# EPICS substitutions: template/evr-cpci-230-ess.substitutions
# Record set for a cPCI-EVR-230
#
# Macros:
#  OBJ = Card name (same as mrmEvrSetupPCI())
#  P and R = System and Device name
#  FEVT = Event link frequency (default 88.0525 MHz)
#
# Record names have the general forms:
#  $(P)$(R=)$(S=:)Signal-SD
#  $(P)$(R=)$(S=:)SubDev-Signal-SD

file "mrmevrbase.template"
{
{P="\$(P)\$(R=)\$(S=:)", PSRC="\$(P)\$(R=)\$(S=:)Src-", PCNT="\$(P)\$(R=)\$(S=:)Cnt-", PLINK="\$(P)\$(R=)\$(S=:)Link-", PRATE="\$(P)\$(R=)\$(S=:)Rate-", PTIME="\$(P)\$(R=)\$(S=:)Time-", OBJ="\$(OBJ)", OBJBUFRX="\$(OBJ):BUFRX", EVNT1HZ="\$(EVNT1HZ=125)", FEVT="\$(FEVT=88.0525)"}
}

file "databuftx.db"
{pattern
{P, OBJ, PROTO}
{"\$(P)\$(R=)\$(S=:)dbus-send-", "\$(OBJ):BUFTX", 1}
}

file "databuftxCtrl.db"
{pattern
{P, OBJ}
{"\$(P)\$(R=)\$(S=:)Link-", "\$(OBJ):BUFTX"}
}

file "mrmevrbufrx.db"
{pattern
{P, OBJ, PROTO}
{"\$(P)\$(R=)\$(S=:)dbus-recv-", \$(OBJ):BUFRX, 0xff00}
}

file "sfp.db"
{
{P="\$(P)\$(R=)\$(S=:)SFP-", PPWR="\$(P)\$(R=)\$(S=:)SFP-Pwr-", PSPEED="\$(P)\$(R=)\$(S=:)SFP-Speed-", PDATE="\$(P)\$(R=)\$(S=:)SFP-Date-", OBJ="\$(OBJ):SFP"}
}

file "evrmap.db"
{pattern
{NAME, OBJ, func, EVT}
{"\$(P)\$(R=)\$(S=:)Evt-Blink0-SP", "\$(OBJ)", Blink, 15}
{"\$(P)\$(R=)\$(S=:)Evt-Blink1-SP", "\$(OBJ)", Blink, 0}
{"\$(P)\$(R=)\$(S=:)Evt-ResetPS-SP","\$(OBJ)", "Reset PS", 123}
}

file "evrevent.db"
{pattern
{EN, OBJ, CODE, EVNT}
{"\$(P)\$(R=)\$(S=:)1hz",  "\$(OBJ)", 0x7d, 125}
{"\$(P)\$(R=)\$(S=:)EvtA", "\$(OBJ)", 10, 10}
{"\$(P)\$(R=)\$(S=:)EvtB", "\$(OBJ)", 11, 11}
{"\$(P)\$(R=)\$(S=:)EvtC", "\$(OBJ)", 12, 12}
{"\$(P)\$(R=)\$(S=:)EvtD", "\$(OBJ)", 13, 13}
{"\$(P)\$(R=)\$(S=:)EvtE", "\$(OBJ)", 14, 14}
{"\$(P)\$(R=)\$(S=:)EvtF", "\$(OBJ)", 15, 15}
{"\$(P)\$(R=)\$(S=:)EvtG", "\$(OBJ)", 16, 16}
{"\$(P)\$(R=)\$(S=:)EvtH", "\$(OBJ)", 17, 17}
}

file "evrscale.db"
{pattern
{IDX, P, SN, OBJ, MAX}
{0, "\$(P)\$(R=)\$(S=:)Link-", "\$(P)\$(R=)\$(S=:)PS$(IDX)-", "\$(OBJ):PS$(IDX)", "0xffffffff"}
{1, "\$(P)\$(R=)\$(S=:)Link-", "\$(P)\$(R=)\$(S=:)PS$(IDX)-", "\$(OBJ):PS$(IDX)", "0xffffffff"}
{2, "\$(P)\$(R=)\$(S=:)Link-", "\$(P)\$(R=)\$(S=:)PS$(IDX)-", "\$(OBJ):PS$(IDX)", "0xffffffff"}
}

file "mrmevrout.db"
{pattern
{ON, ONSRC, OBJ, DESC}
{"\$(P)\$(R=)\$(S=:)OutInt-", "\$(P)\$(R=)\$(S=:)OutInt-Src-", "\$(OBJ):Int", "Internal"}
{"\$(P)\$(R=)\$(S=:)OutFPUV0-", "\$(P)\$(R=)\$(S=:)OutFPUV0-Src-", "\$(OBJ):FrontUnivOut0", "UNIV0"}
{"\$(P)\$(R=)\$(S=:)OutFPUV1-", "\$(P)\$(R=)\$(S=:)OutFPUV1-Src-", "\$(OBJ):FrontUnivOut1", "UNIV1"}
{"\$(P)\$(R=)\$(S=:)OutFPUV2-", "\$(P)\$(R=)\$(S=:)OutFPUV2-Src-", "\$(OBJ):FrontUnivOut2", "UNIV2"}
{"\$(P)\$(R=)\$(S=:)OutFPUV3-", "\$(P)\$(R=)\$(S=:)OutFPUV3-Src-", "\$(OBJ):FrontUnivOut3", "UNIV3"}
}

file "mrmevroutint.db"
{{
    ON="\$(P)\$(R=)\$(S=:)OutInt-", OBJ="\$(OBJ)"
}}

# Pulse generators w/o a prescaler set NOPS=1
file "evrpulser.db"
{pattern
{PID, P, PLINK, PN, PNDELAY, PNWIDTH, OBJ, DMAX, WMAX, PMAX, NOPS}
{0, "\$(P)\$(R=)\$(S=:)", "\$(P)\$(R=)\$(S=:)Link-", "\$(P)\$(R=)\$(S=:)DlyGen$(PID)-", "\$(P)\$(R=)\$(S=:)DlyGen$(PID)-Delay-", "\$(P)\$(R=)\$(S=:)DlyGen$(PID)-Width-", "\$(OBJ):Pul$(PID)", "0xffffffff", "0xffffffff", "0xffff", 0}
{1, "\$(P)\$(R=)\$(S=:)", "\$(P)\$(R=)\$(S=:)Link-", "\$(P)\$(R=)\$(S=:)DlyGen$(PID)-", "\$(P)\$(R=)\$(S=:)DlyGen$(PID)-Delay-", "\$(P)\$(R=)\$(S=:)DlyGen$(PID)-Width-", "\$(OBJ):Pul$(PID)", "0xffffffff", "0xffffffff", "0xffff", 0}
{2, "\$(P)\$(R=)\$(S=:)", "\$(P)\$(R=)\$(S=:)Link-", "\$(P)\$(R=)\$(S=:)DlyGen$(PID)-", "\$(P)\$(R=)\$(S=:)DlyGen$(PID)-Delay-", "\$(P)\$(R=)\$(S=:)DlyGen$(PID)-Width-", "\$(OBJ):Pul$(PID)", "0xffffffff", "0xffffffff", "0xffff", 0}
{3, "\$(P)\$(R=)\$(S=:)", "\$(P)\$(R=)\$(S=:)Link-", "\$(P)\$(R=)\$(S=:)DlyGen$(PID)-", "\$(P)\$(R=)\$(S=:)DlyGen$(PID)-Delay-", "\$(P)\$(R=)\$(S=:)DlyGen$(PID)-Width-", "\$(OBJ):Pul$(PID)", "0xffffffff", "0xffffffff", "0xffff", 0}
{4, "\$(P)\$(R=)\$(S=:)", "\$(P)\$(R=)\$(S=:)Link-", "\$(P)\$(R=)\$(S=:)DlyGen$(PID)-", "\$(P)\$(R=)\$(S=:)DlyGen$(PID)-Delay-", "\$(P)\$(R=)\$(S=:)DlyGen$(PID)-Width-", "\$(OBJ):Pul$(PID)", "0xffffffff", "0xffff", "1", 1}
{5, "\$(P)\$(R=)\$(S=:)", "\$(P)\$(R=)\$(S=:)Link-", "\$(P)\$(R=)\$(S=:)DlyGen$(PID)-", "\$(P)\$(R=)\$(S=:)DlyGen$(PID)-Delay-", "\$(P)\$(R=)\$(S=:)DlyGen$(PID)-Width-", "\$(OBJ):Pul$(PID)", "0xffffffff", "0xffff", "1", 1}
{6, "\$(P)\$(R=)\$(S=:)", "\$(P)\$(R=)\$(S=:)Link-", "\$(P)\$(R=)\$(S=:)DlyGen$(PID)-", "\$(P)\$(R=)\$(S=:)DlyGen$(PID)-Delay-", "\$(P)\$(R=)\$(S=:)DlyGen$(PID)-Width-", "\$(OBJ):Pul$(PID)", "0xffffffff", "0xffff", "1", 1}
{7, "\$(P)\$(R=)\$(S=:)", "\$(P)\$(R=)\$(S=:)Link-", "\$(P)\$(R=)\$(S=:)DlyGen$(PID)-", "\$(P)\$(R=)\$(S=:)DlyGen$(PID)-Delay-", "\$(P)\$(R=)\$(S=:)DlyGen$(PID)-Width-", "\$(OBJ):Pul$(PID)", "0xffffffff", "0xffff", "1", 1}
{8, "\$(P)\$(R=)\$(S=:)", "\$(P)\$(R=)\$(S=:)Link-", "\$(P)\$(R=)\$(S=:)DlyGen$(PID)-", "\$(P)\$(R=)\$(S=:)DlyGen$(PID)-Delay-", "\$(P)\$(R=)\$(S=:)DlyGen$(PID)-Width-", "\$(OBJ):Pul$(PID)", "0xffffffff", "0xffff", "1", 1}
{9, "\$(P)\$(R=)\$(S=:)", "\$(P)\$(R=)\$(S=:)Link-", "\$(P)\$(R=)\$(S=:)DlyGen$(PID)-", "\$(P)\$(R=)\$(S=:)DlyGen$(PID)-Delay-", "\$(P)\$(R=)\$(S=:)DlyGen$(PID)-Width-", "\$(OBJ):Pul$(PID)", "0xffffffff", "0xffff", "1", 1}
}

# Default to 3 possible trigger mappings per pulser
file "evrpulsermap.db"
{pattern
{PID, NAME, OBJ, F, EVT}
{0, "\$(P)\$(R=)\$(S=:)DlyGen$(PID)-Evt-Trig0-SP", "\$(OBJ):Pul$(PID)", Trig, 0}
{0, "\$(P)\$(R=)\$(S=:)DlyGen$(PID)-Evt-Trig1-SP", "\$(OBJ):Pul$(PID)", Trig, 0}
{0, "\$(P)\$(R=)\$(S=:)DlyGen$(PID)-Evt-Trig2-SP", "\$(OBJ):Pul$(PID)", Trig, 0}
{1, "\$(P)\$(R=)\$(S=:)DlyGen$(PID)-Evt-Trig0-SP", "\$(OBJ):Pul$(PID)", Trig, 0}
{1, "\$(P)\$(R=)\$(S=:)DlyGen$(PID)-Evt-Trig1-SP", "\$(OBJ):Pul$(PID)", Trig, 0}
{1, "\$(P)\$(R=)\$(S=:)DlyGen$(PID)-Evt-Trig2-SP", "\$(OBJ):Pul$(PID)", Trig, 0}
{2, "\$(P)\$(R=)\$(S=:)DlyGen$(PID)-Evt-Trig0-SP", "\$(OBJ):Pul$(PID)", Trig, 0}
{2, "\$(P)\$(R=)\$(S=:)DlyGen$(PID)-Evt-Trig1-SP", "\$(OBJ):Pul$(PID)", Trig, 0}
{2, "\$(P)\$(R=)\$(S=:)DlyGen$(PID)-Evt-Trig2-SP", "\$(OBJ):Pul$(PID)", Trig, 0}
{3, "\$(P)\$(R=)\$(S=:)DlyGen$(PID)-Evt-Trig0-SP", "\$(OBJ):Pul$(PID)", Trig, 0}
{3, "\$(P)\$(R=)\$(S=:)DlyGen$(PID)-Evt-Trig1-SP", "\$(OBJ):Pul$(PID)", Trig, 0}
{3, "\$(P)\$(R=)\$(S=:)DlyGen$(PID)-Evt-Trig2-SP", "\$(OBJ):Pul$(PID)", Trig, 0}
{4, "\$(P)\$(R=)\$(S=:)DlyGen$(PID)-Evt-Trig0-SP", "\$(OBJ):Pul$(PID)", Trig, 0}
{4, "\$(P)\$(R=)\$(S=:)DlyGen$(PID)-Evt-Trig1-SP", "\$(OBJ):Pul$(PID)", Trig, 0}
{4, "\$(P)\$(R=)\$(S=:)DlyGen$(PID)-Evt-Trig2-SP", "\$(OBJ):Pul$(PID)", Trig, 0}
{5, "\$(P)\$(R=)\$(S=:)DlyGen$(PID)-Evt-Trig0-SP", "\$(OBJ):Pul$(PID)", Trig, 0}
{5, "\$(P)\$(R=)\$(S=:)DlyGen$(PID)-Evt-Trig1-SP", "\$(OBJ):Pul$(PID)", Trig, 0}
{5, "\$(P)\$(R=)\$(S=:)DlyGen$(PID)-Evt-Trig2-SP", "\$(OBJ):Pul$(PID)", Trig, 0}
{6, "\$(P)\$(R=)\$(S=:)DlyGen$(PID)-Evt-Trig0-SP", "\$(OBJ):Pul$(PID)", Trig, 0}
{6, "\$(P)\$(R=)\$(S=:)DlyGen$(PID)-Evt-Trig1-SP", "\$(OBJ):Pul$(PID)", Trig, 0}
{6, "\$(P)\$(R=)\$(S=:)DlyGen$(PID)-Evt-Trig2-SP", "\$(OBJ):Pul$(PID)", Trig, 0}
{7, "\$(P)\$(R=)\$(S=:)DlyGen$(PID)-Evt-Trig0-SP", "\$(OBJ):Pul$(PID)", Trig, 0}
{7, "\$(P)\$(R=)\$(S=:)DlyGen$(PID)-Evt-Trig1-SP", "\$(OBJ):Pul$(PID)", Trig, 0}
{7, "\$(P)\$(R=)\$(S=:)DlyGen$(PID)-Evt-Trig2-SP", "\$(OBJ):Pul$(PID)", Trig, 0}
{8, "\$(P)\$(R=)\$(S=:)DlyGen$(PID)-Evt-Trig0-SP", "\$(OBJ):Pul$(PID)", Trig, 0}
{8, "\$(P)\$(R=)\$(S=:)DlyGen$(PID)-Evt-Trig1-SP", "\$(OBJ):Pul$(PID)", Trig, 0}
{8, "\$(P)\$(R=)\$(S=:)DlyGen$(PID)-Evt-Trig2-SP", "\$(OBJ):Pul$(PID)", Trig, 0}
{9, "\$(P)\$(R=)\$(S=:)DlyGen$(PID)-Evt-Trig0-SP", "\$(OBJ):Pul$(PID)", Trig, 0}
{9, "\$(P)\$(R=)\$(S=:)DlyGen$(PID)-Evt-Trig1-SP", "\$(OBJ):Pul$(PID)", Trig, 0}
{9, "\$(P)\$(R=)\$(S=:)DlyGen$(PID)-Evt-Trig2-SP", "\$(OBJ):Pul$(PID)", Trig, 0}
}

file "evrin.db"
{pattern
{IN, INTRIG, INCODE, OBJ, DESC}
{"\$(P)\$(R=)\$(S=:)In0-", "\$(P)\$(R=)\$(S=:)In0-Trig-", "\$(P)\$(R=)\$(S=:)In0-Code-", "\$(OBJ):FPIn0", "IN0 (TTL)"}
{"\$(P)\$(R=)\$(S=:)In1-", "\$(P)\$(R=)\$(S=:)In1-Trig-", "\$(P)\$(R=)\$(S=:)In1-Code-", "\$(OBJ):FPIn1", "IN1 (TTL)"}
}
